// TIA Portal V17 export
// export: Created 2024-09-27T21:44:58.5464654Z, ExportSetting WithDefaults, DisplayName Totally Integrated Automation Portal, DisplayVersion V17, DisplayName TIA Portal Openness, DisplayVersion V17, DisplayName TIA Portal Version Control Interface, DisplayVersion V17, DisplayName STEP 7 Professional, DisplayVersion V17, DisplayName STEP 7 Safety, DisplayVersion V17, DisplayName WinCC Professional, DisplayVersion V17
DATA_BLOCK "reference_values"   // DB26
{ S7_Optimized_Access := 'TRUE' }
VERSION : 0.1
// stored: AutoNumber true, DBAccessibleFromOPCUA true, IsOnlyStoredInLoadMemory false, IsRetainMemResEnabled false, IsWriteProtectedInAS false, MemoryReserve 100
   VAR RETAIN
      ref1_takt_stołu : Time := T#7S;
      ref1_pred_stolu : Real := 50.0;
      ref1_czas_ssania : Time := T#1S;
      ref1_czas_przedmuchu : Time := T#1S;
      ref1_delay_sił_zag_dół : Time := T#100MS;
   END_VAR
   VAR
      ref1_delay_sił_odb_stol : Time := T#1S;
   END_VAR
BEGIN
END_DATA_BLOCK
